FUNCTION_BLOCK FB_HaltNC_TestDouble IMPLEMENTS  I_Halt
VAR_INPUT
END_VAR
VAR_OUTPUT
END_VAR
VAR
END_VAR

{warning 'Add property implementation'}
PROPERTY Aborted : BOOL
GET
END_GET
END_PROPERTY

{warning 'Add property implementation'}
PROPERTY Active : BOOL
GET
END_GET
END_PROPERTY

{warning 'Add property implementation'}
PROPERTY Busy : BOOL
GET
END_GET
END_PROPERTY

{warning 'Add property implementation'}
PROPERTY CommandHalt : BOOL
SET
END_SET
END_PROPERTY

{warning 'Add property implementation'}
PROPERTY Done : BOOL
GET
END_GET
END_PROPERTY

{warning 'Add property implementation'}
PROPERTY Error : BOOL
GET
END_GET
END_PROPERTY

{warning 'Add property implementation'}
PROPERTY ErrorID : UDINT
GET
END_GET
END_PROPERTY

{warning 'Add method implementation '}
METHOD Halt
VAR_INPUT
    Deceleration	: LREAL := 0;
    Jerk	: LREAL := 0;
    BufferMode	: MC_BufferMode := .MC_BufferMode.MC_Aborting;
END_VAR
END_METHOD

{warning 'Add property implementation'}
PROPERTY Message : T_MAXSTRING
GET
END_GET
END_PROPERTY

END_FUNCTION_BLOCK

(* stored: Version 1.1.0.1
   POU FB_HaltNC_TestDouble: Id {f9b66d85-7bb4-402b-9f8b-2a0adea12002}, SpecialFunc None
   Property Aborted: Id {93737e43-fd27-4bc9-ba9b-223268f682f3}
   Get Get: Id {fef0ec11-61d3-4e40-a4b0-f1ca0db49a20}
   Property Active: Id {2b37f2d8-d99f-4670-9e2e-6850dbfbedbf}
   Get Get: Id {8e8336dc-0a95-41af-9c36-72bf717dcc13}
   Property Busy: Id {034fa069-6878-4483-aee8-f3158caaf3b6}
   Get Get: Id {b063851c-4493-4d17-ae35-c9062adea97f}
   Property CommandHalt: Id {086e355b-6176-40fc-aa49-523c080ad882}
   Set Set: Id {5538a0dc-0e1c-45bd-acb0-31a7a9925af1}
   Property Done: Id {a4f4af90-5ae1-4477-b229-6a6b6705b3dd}
   Get Get: Id {b1cf0137-23e5-4693-b43b-e15d2c9344c1}
   Property Error: Id {cc116eda-d8d1-4a1d-82e6-92ac9919db6f}
   Get Get: Id {5fcda727-bdc7-41fc-9341-c44594191003}
   Property ErrorID: Id {d686636c-b18c-4f6b-855d-6b987cd35849}
   Get Get: Id {70e690d0-ec33-418c-8670-d56a804c91a0}
   Method Halt: Id {6b0a130f-519e-48ff-97cd-c37fb031ebbf}
   Property Message: Id {9dd1b35c-115d-4a93-bec5-c49881409ad8}
   Get Get: Id {4afe19f6-0305-4dc4-be85-e22907dd5c3a} *)
